{attribute 'qualified_only'}
{attribute 'strict'}
TYPE EProductTypes :
(
	none := 0,
	unknown := 1,
	
	white := 2,
	black := 3,
	metal := 4
) UINT;
END_TYPE

(* stored: Version 1.1.0.1, ProductVersion 3.1.4024.9
   DUT EProductTypes: Id {fab6ce6e-9d29-46b5-90af-c1f60090c070} *)
